(* Logix 5000 project; controller Universal_Device_Info_AOI_V0_1 vendor 1 type 14 code 176 rev 32.11; software revision 32.00; part 10 of 11 *)
(* tags used below, declared in another part *)
   Port : INT;
   Common_Data : Turck_IOLink_Common_Data;
   Write_Application_Specific_Tag : BOOL;
   Universal_IOLink_Info : Universal_IOLink_Info;
   StartupDone : BOOL;
   Done : DINT;
   Error : DINT;
   Active : DINT;
   Pending : DINT;
   Pending_or_Active : DINT;
   MyTicketNum : DINT[32];
   Read_ONS : DINT;
   ReadRequest : DINT;
   Read : DINT;
   DoneCount : DINT;
   Status : DINT;
   ErrorCount : DINT;
   Update_Data : BOOL;
   Write_ONS : DINT;
   WriteRequest : DINT;
(* Universal_Device_Info, continued *)

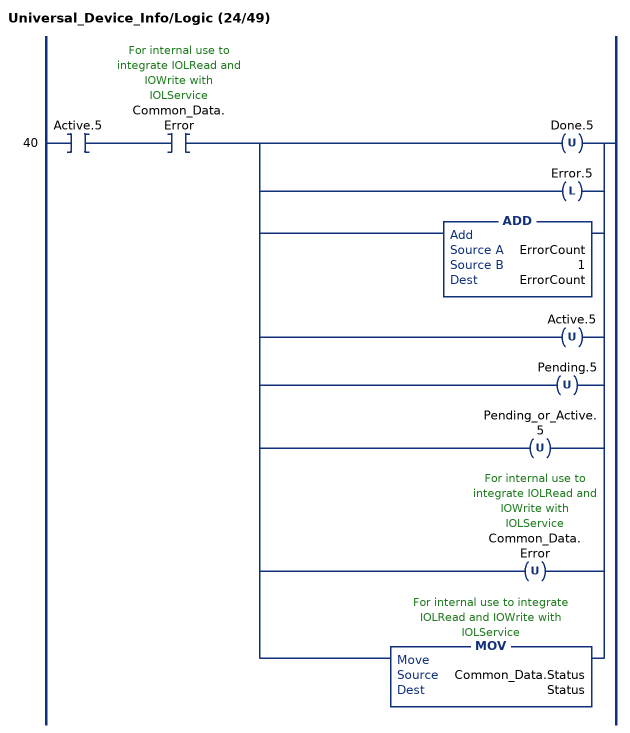
   [picture p67: Universal_Device_Info/Logic rungs 40-40]
   40: XIC(Active.5)XIC(Common_Data.Error)[OTU(Done.5) ,OTL(Error.5) ,ADD(ErrorCount,1,ErrorCount) ,OTU(Active.5) ,OTU(Pending.5) ,OTU(Pending_or_Active.5) ,OTU(Common_Data.Error) ,MOV(Common_Data.Status,Status) ];
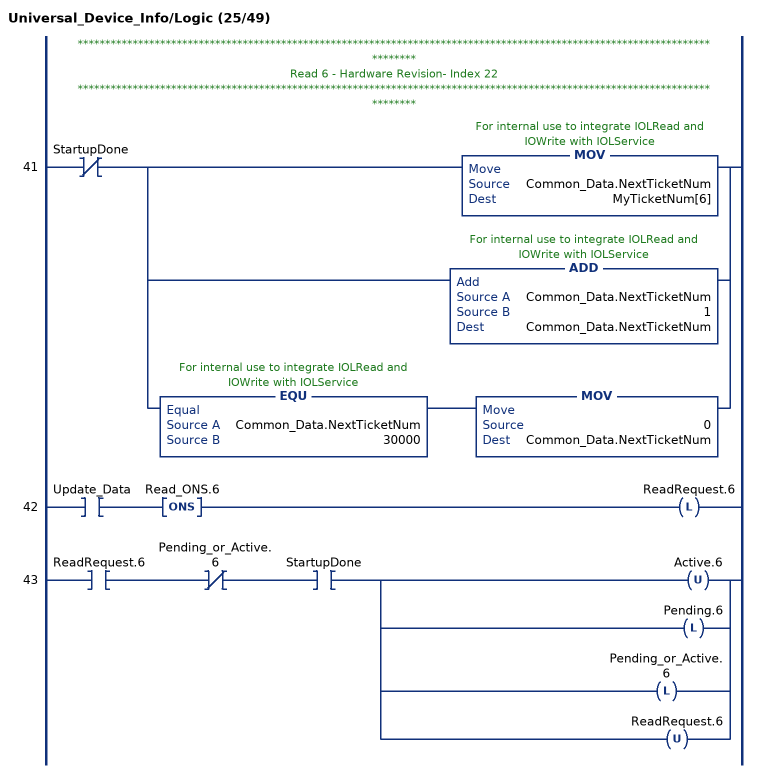
   // ***************************************************************************************************************************
   // Read 6 - Hardware Revision- Index 22
   // ***************************************************************************************************************************
   41: XIO(StartupDone)[MOV(Common_Data.NextTicketNum,MyTicketNum[6]) ,ADD(Common_Data.NextTicketNum,1,Common_Data.NextTicketNum) ,EQU(Common_Data.NextTicketNum,30000) MOV(0,Common_Data.NextTicketNum) ];
   42: XIC(Update_Data)ONS(Read_ONS.6)OTL(ReadRequest.6);
   43: XIC(ReadRequest.6)XIO(Pending_or_Active.6)XIC(StartupDone)[OTU(Active.6) ,OTL(Pending.6) ,OTL(Pending_or_Active.6) ,OTU(ReadRequest.6) ];
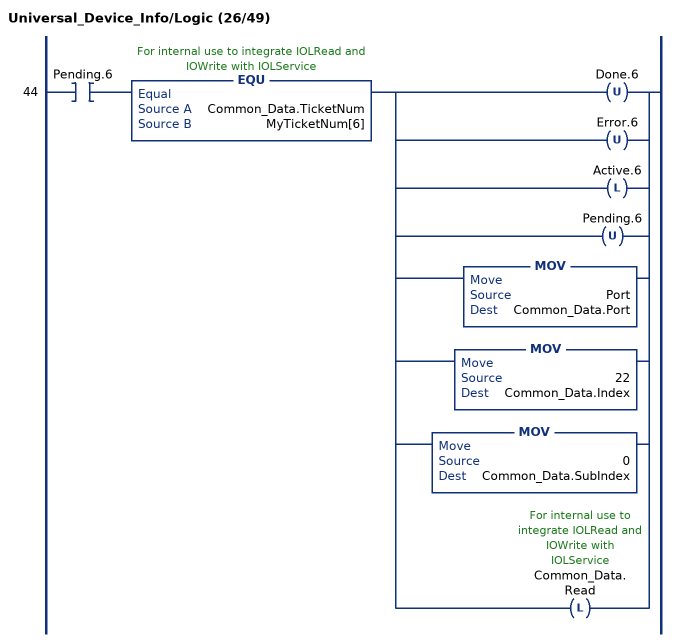
   44: XIC(Pending.6)EQU(Common_Data.TicketNum,MyTicketNum[6])[OTU(Done.6) ,OTU(Error.6) ,OTL(Active.6) ,OTU(Pending.6) ,MOV(Port,Common_Data.Port) ,MOV(22,Common_Data.Index) ,MOV(0,Common_Data.SubIndex) ,OTL(Common_Data.Read) ];
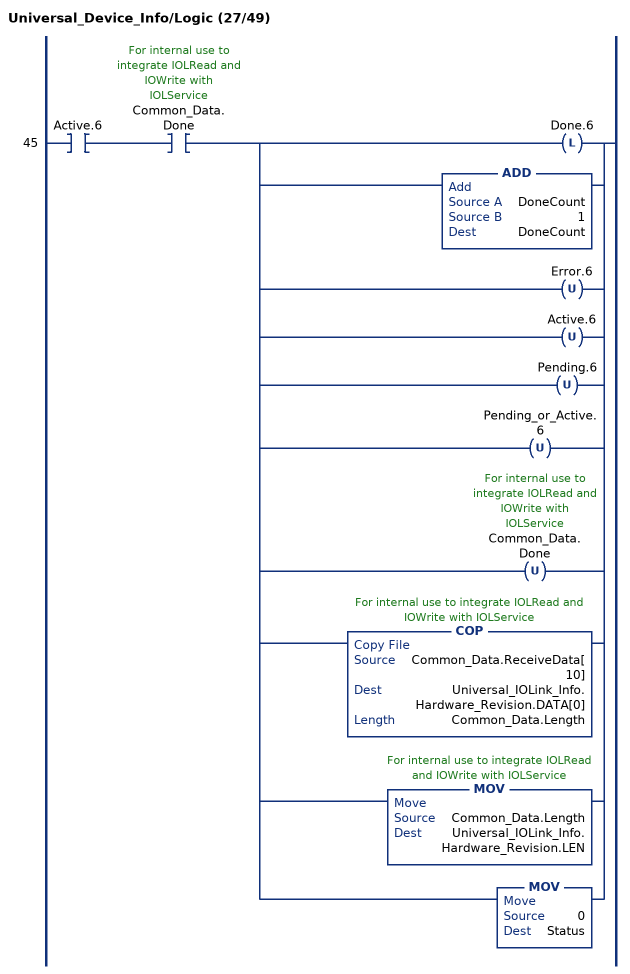
   45: XIC(Active.6)XIC(Common_Data.Done)[OTL(Done.6) ,ADD(DoneCount,1,DoneCount) ,OTU(Error.6) ,OTU(Active.6) ,OTU(Pending.6) ,OTU(Pending_or_Active.6) ,OTU(Common_Data.Done) ,COP(Common_Data.ReceiveData[10],Universal_IOLink_Info.Hardware_Revision.DATA[0],Common_Data.Length) ,MOV(Common_Data.Length,Universal_IOLink_Info.Hardware_Revision.LEN) ,MOV(0,Status) ];
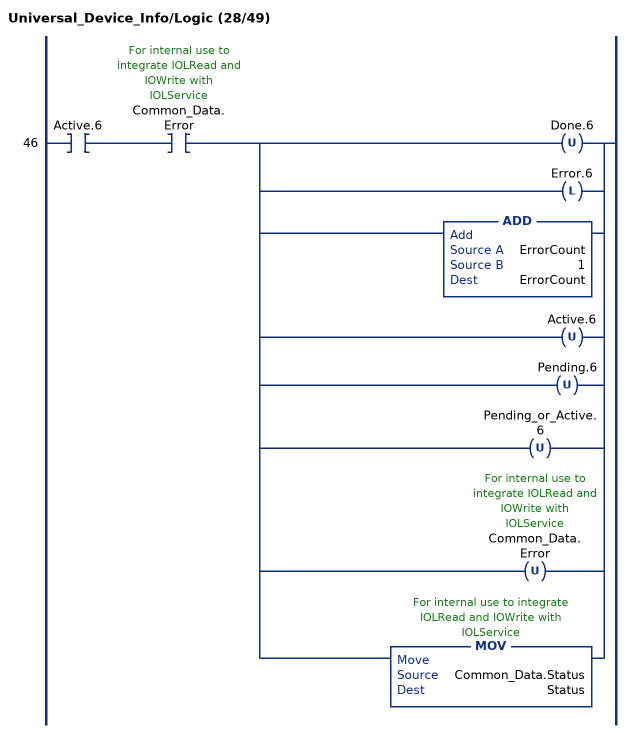
   46: XIC(Active.6)XIC(Common_Data.Error)[OTU(Done.6) ,OTL(Error.6) ,ADD(ErrorCount,1,ErrorCount) ,OTU(Active.6) ,OTU(Pending.6) ,OTU(Pending_or_Active.6) ,OTU(Common_Data.Error) ,MOV(Common_Data.Status,Status) ];
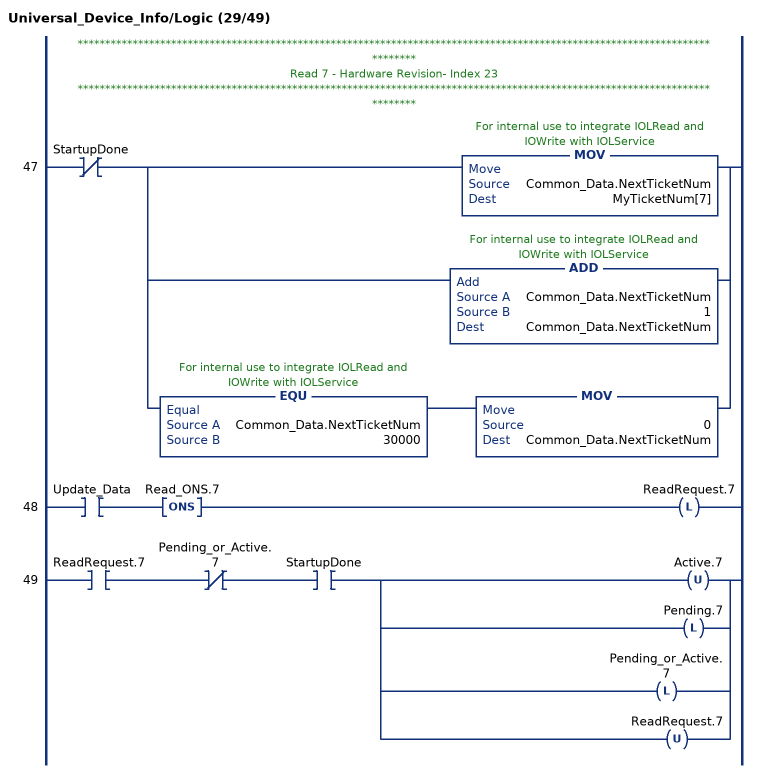
   // ***************************************************************************************************************************
   // Read 7 - Hardware Revision- Index 23
   // ***************************************************************************************************************************
   47: XIO(StartupDone)[MOV(Common_Data.NextTicketNum,MyTicketNum[7]) ,ADD(Common_Data.NextTicketNum,1,Common_Data.NextTicketNum) ,EQU(Common_Data.NextTicketNum,30000) MOV(0,Common_Data.NextTicketNum) ];
   48: XIC(Update_Data)ONS(Read_ONS.7)OTL(ReadRequest.7);
   49: XIC(ReadRequest.7)XIO(Pending_or_Active.7)XIC(StartupDone)[OTU(Active.7) ,OTL(Pending.7) ,OTL(Pending_or_Active.7) ,OTU(ReadRequest.7) ];
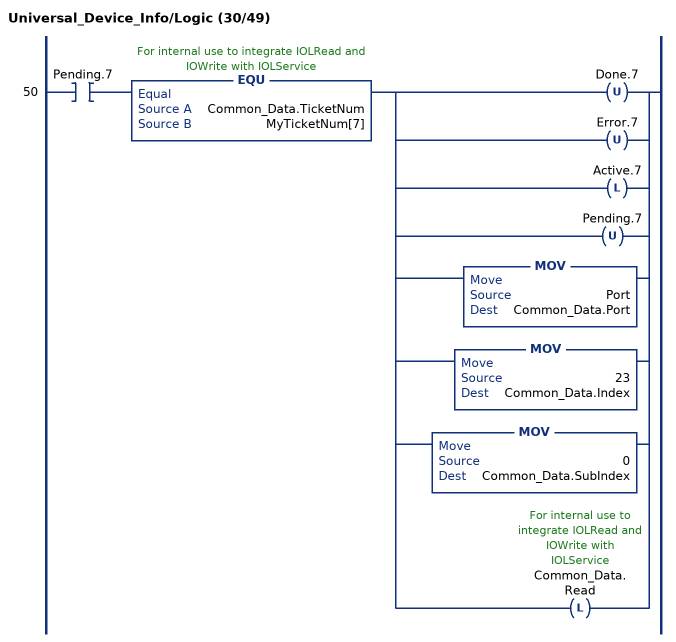
   50: XIC(Pending.7)EQU(Common_Data.TicketNum,MyTicketNum[7])[OTU(Done.7) ,OTU(Error.7) ,OTL(Active.7) ,OTU(Pending.7) ,MOV(Port,Common_Data.Port) ,MOV(23,Common_Data.Index) ,MOV(0,Common_Data.SubIndex) ,OTL(Common_Data.Read) ];
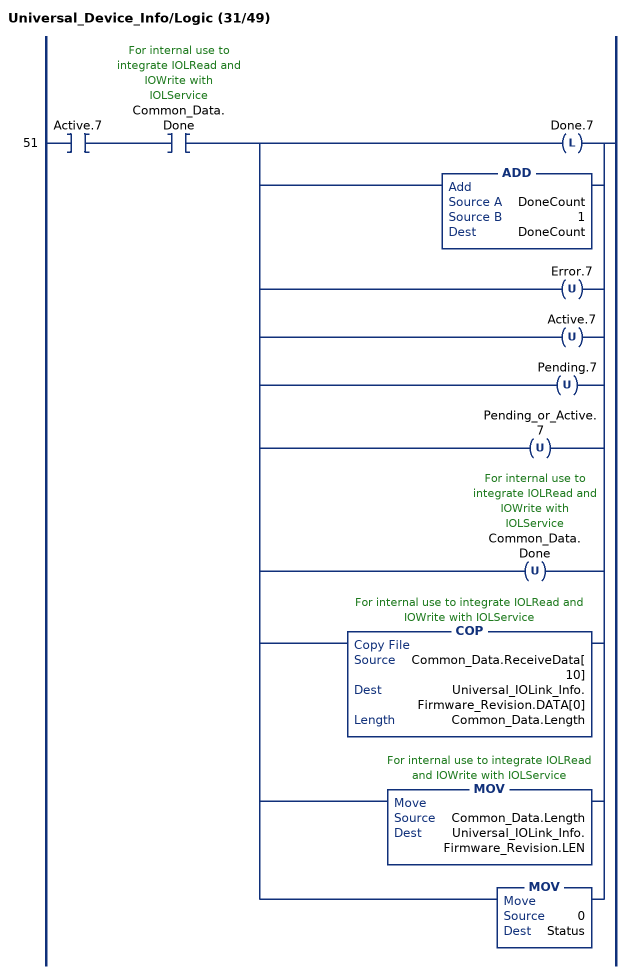
   51: XIC(Active.7)XIC(Common_Data.Done)[OTL(Done.7) ,ADD(DoneCount,1,DoneCount) ,OTU(Error.7) ,OTU(Active.7) ,OTU(Pending.7) ,OTU(Pending_or_Active.7) ,OTU(Common_Data.Done) ,COP(Common_Data.ReceiveData[10],Universal_IOLink_Info.Firmware_Revision.DATA[0],Common_Data.Length) ,MOV(Common_Data.Length,Universal_IOLink_Info.Firmware_Revision.LEN) ,MOV(0,Status) ];
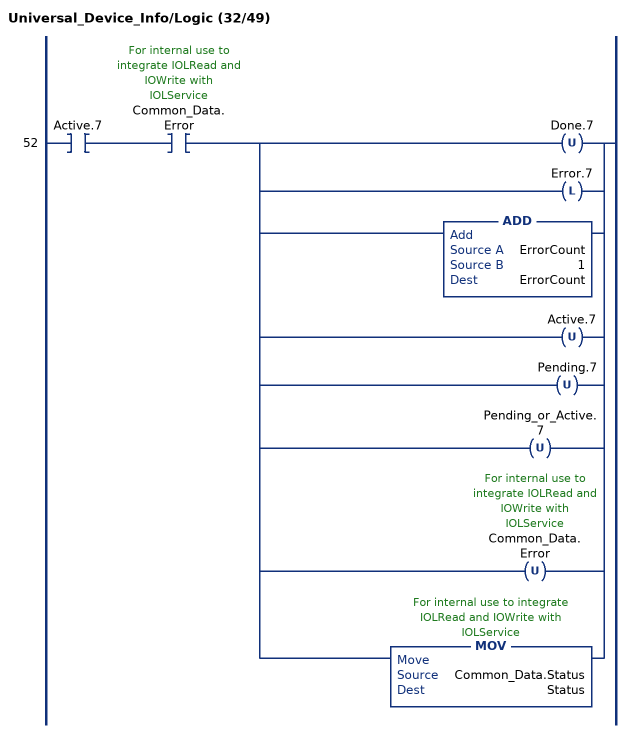
   52: XIC(Active.7)XIC(Common_Data.Error)[OTU(Done.7) ,OTL(Error.7) ,ADD(ErrorCount,1,ErrorCount) ,OTU(Active.7) ,OTU(Pending.7) ,OTU(Pending_or_Active.7) ,OTU(Common_Data.Error) ,MOV(Common_Data.Status,Status) ];
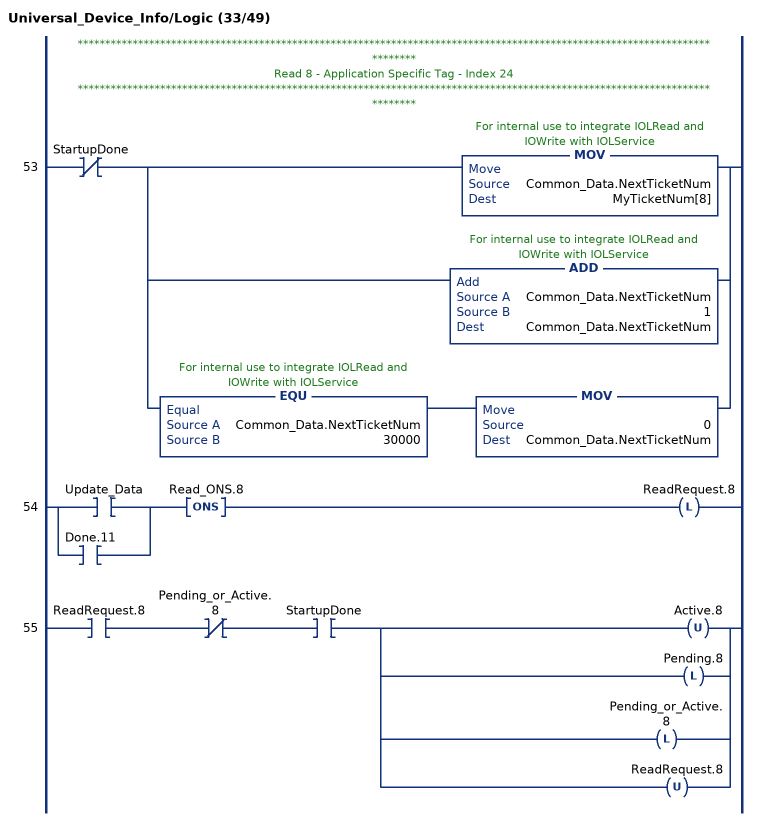
   // ***************************************************************************************************************************
   // Read 8 - Application Specific Tag - Index 24
   // ***************************************************************************************************************************
   53: XIO(StartupDone)[MOV(Common_Data.NextTicketNum,MyTicketNum[8]) ,ADD(Common_Data.NextTicketNum,1,Common_Data.NextTicketNum) ,EQU(Common_Data.NextTicketNum,30000) MOV(0,Common_Data.NextTicketNum) ];
   54: [XIC(Update_Data) ,XIC(Done.11) ]ONS(Read_ONS.8)OTL(ReadRequest.8);
   55: XIC(ReadRequest.8)XIO(Pending_or_Active.8)XIC(StartupDone)[OTU(Active.8) ,OTL(Pending.8) ,OTL(Pending_or_Active.8) ,OTU(ReadRequest.8) ];
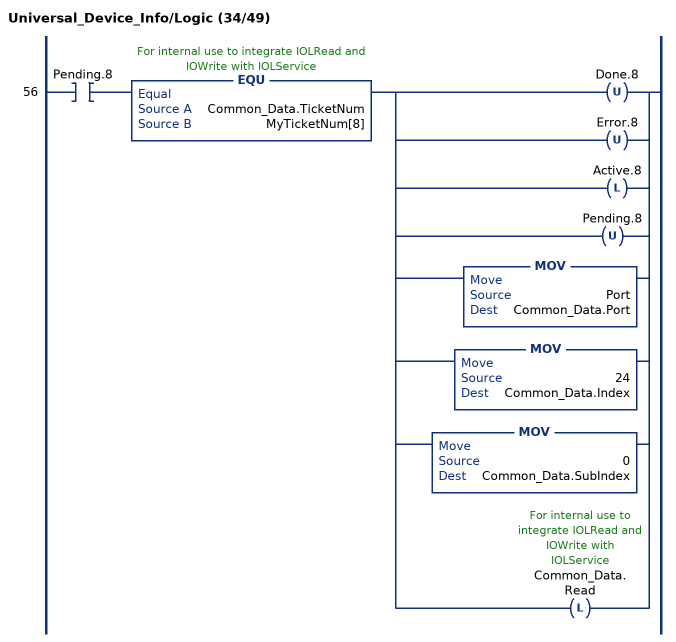
   56: XIC(Pending.8)EQU(Common_Data.TicketNum,MyTicketNum[8])[OTU(Done.8) ,OTU(Error.8) ,OTL(Active.8) ,OTU(Pending.8) ,MOV(Port,Common_Data.Port) ,MOV(24,Common_Data.Index) ,MOV(0,Common_Data.SubIndex) ,OTL(Common_Data.Read) ];
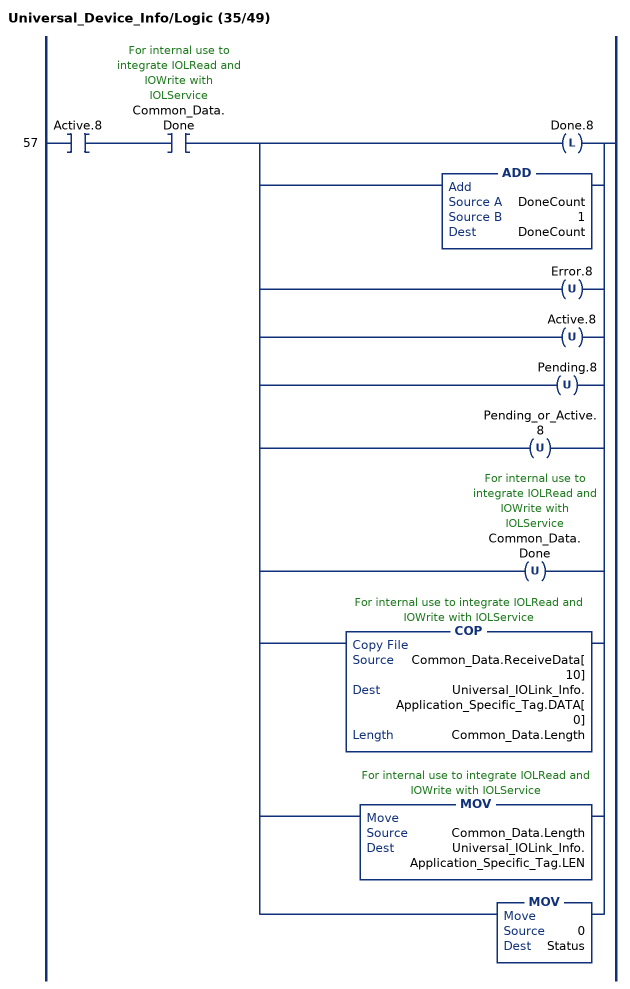
   57: XIC(Active.8)XIC(Common_Data.Done)[OTL(Done.8) ,ADD(DoneCount,1,DoneCount) ,OTU(Error.8) ,OTU(Active.8) ,OTU(Pending.8) ,OTU(Pending_or_Active.8) ,OTU(Common_Data.Done) ,COP(Common_Data.ReceiveData[10],Universal_IOLink_Info.Application_Specific_Tag.DATA[0],Common_Data.Length) ,MOV(Common_Data.Length,Universal_IOLink_Info.Application_Specific_Tag.LEN) ,MOV(0,Status) ];
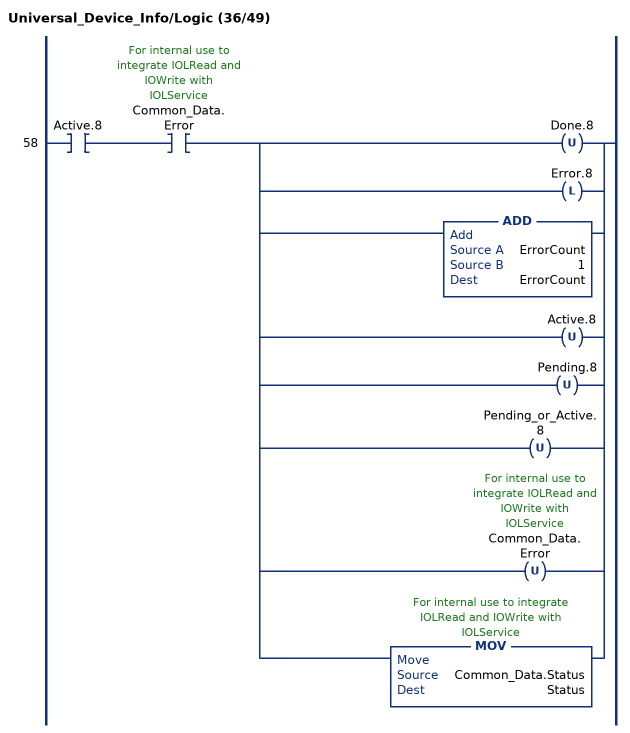
   58: XIC(Active.8)XIC(Common_Data.Error)[OTU(Done.8) ,OTL(Error.8) ,ADD(ErrorCount,1,ErrorCount) ,OTU(Active.8) ,OTU(Pending.8) ,OTU(Pending_or_Active.8) ,OTU(Common_Data.Error) ,MOV(Common_Data.Status,Status) ];
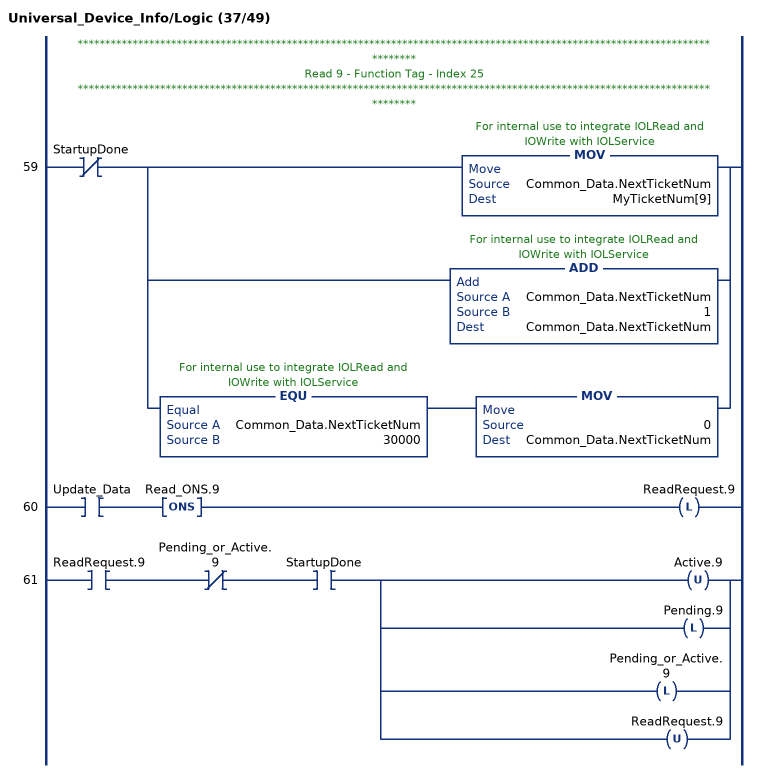
   // ***************************************************************************************************************************
   // Read 9 - Function Tag - Index 25
   // ***************************************************************************************************************************
   59: XIO(StartupDone)[MOV(Common_Data.NextTicketNum,MyTicketNum[9]) ,ADD(Common_Data.NextTicketNum,1,Common_Data.NextTicketNum) ,EQU(Common_Data.NextTicketNum,30000) MOV(0,Common_Data.NextTicketNum) ];
   60: XIC(Update_Data)ONS(Read_ONS.9)OTL(ReadRequest.9);
   61: XIC(ReadRequest.9)XIO(Pending_or_Active.9)XIC(StartupDone)[OTU(Active.9) ,OTL(Pending.9) ,OTL(Pending_or_Active.9) ,OTU(ReadRequest.9) ];
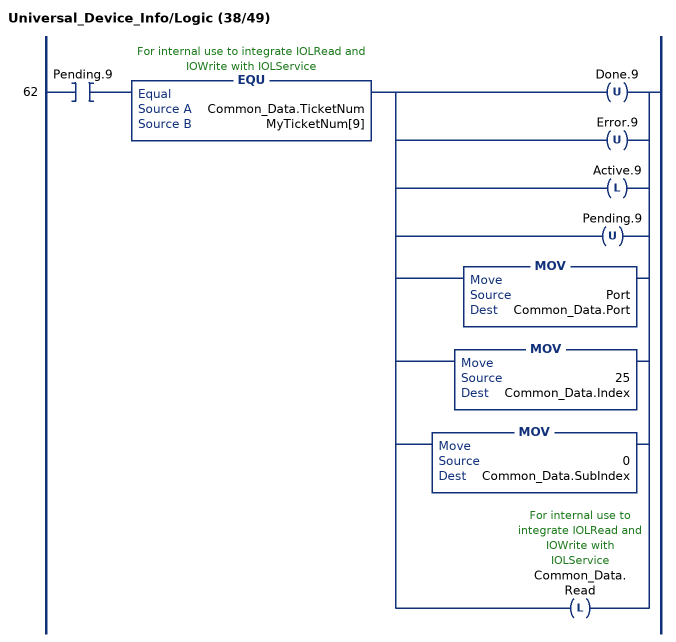
   62: XIC(Pending.9)EQU(Common_Data.TicketNum,MyTicketNum[9])[OTU(Done.9) ,OTU(Error.9) ,OTL(Active.9) ,OTU(Pending.9) ,MOV(Port,Common_Data.Port) ,MOV(25,Common_Data.Index) ,MOV(0,Common_Data.SubIndex) ,OTL(Common_Data.Read) ];
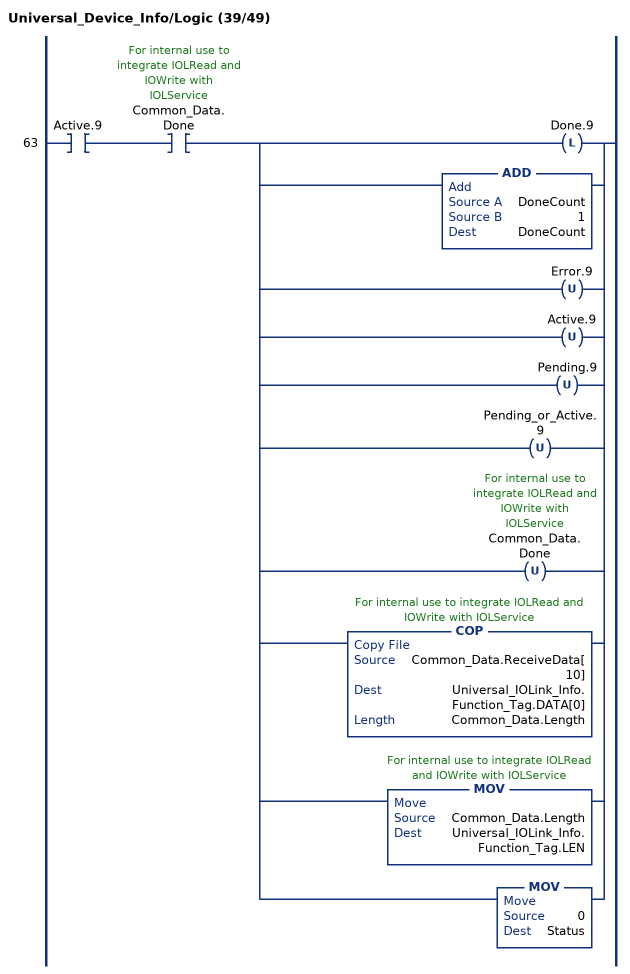
   63: XIC(Active.9)XIC(Common_Data.Done)[OTL(Done.9) ,ADD(DoneCount,1,DoneCount) ,OTU(Error.9) ,OTU(Active.9) ,OTU(Pending.9) ,OTU(Pending_or_Active.9) ,OTU(Common_Data.Done) ,COP(Common_Data.ReceiveData[10],Universal_IOLink_Info.Function_Tag.DATA[0],Common_Data.Length) ,MOV(Common_Data.Length,Universal_IOLink_Info.Function_Tag.LEN) ,MOV(0,Status) ];
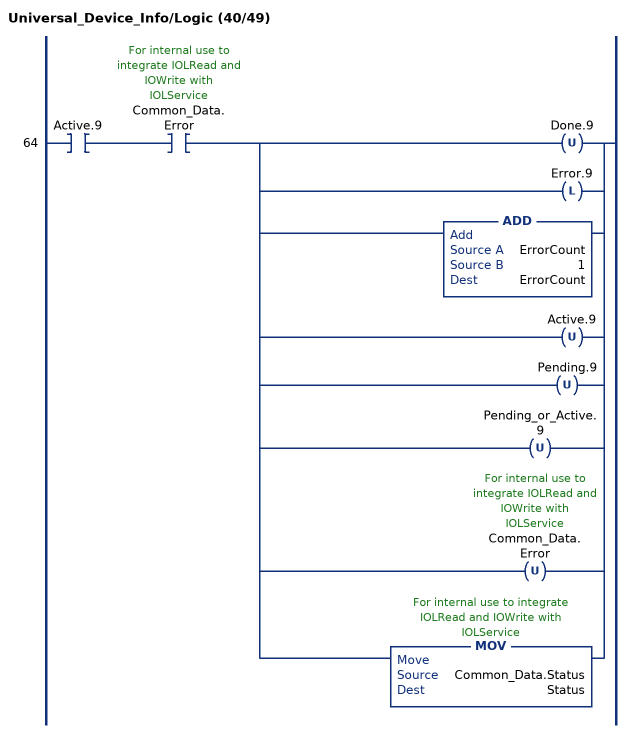
   64: XIC(Active.9)XIC(Common_Data.Error)[OTU(Done.9) ,OTL(Error.9) ,ADD(ErrorCount,1,ErrorCount) ,OTU(Active.9) ,OTU(Pending.9) ,OTU(Pending_or_Active.9) ,OTU(Common_Data.Error) ,MOV(Common_Data.Status,Status) ];
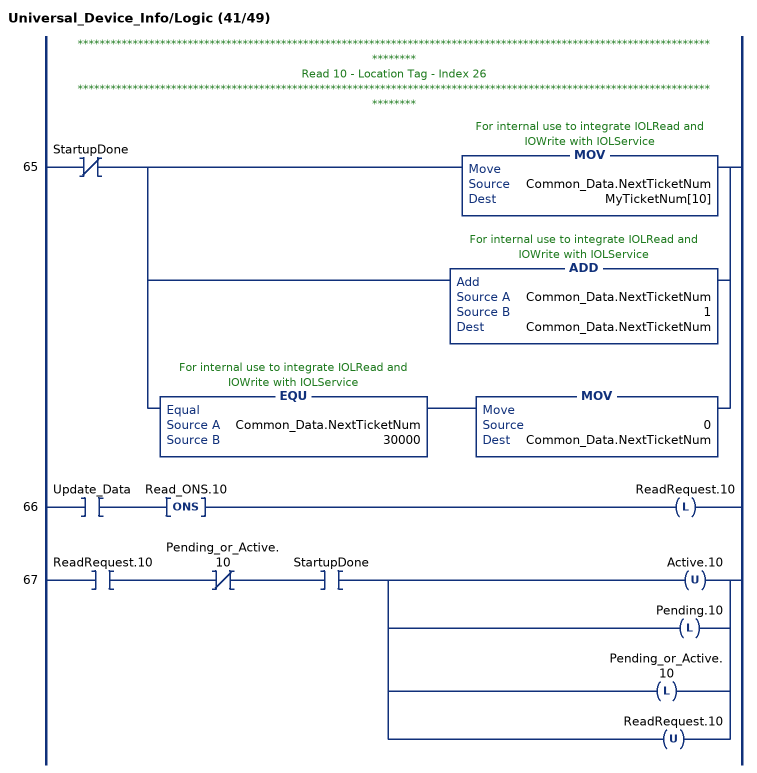
   // ***************************************************************************************************************************
   // Read 10 - Location Tag - Index 26
   // ***************************************************************************************************************************
   65: XIO(StartupDone)[MOV(Common_Data.NextTicketNum,MyTicketNum[10]) ,ADD(Common_Data.NextTicketNum,1,Common_Data.NextTicketNum) ,EQU(Common_Data.NextTicketNum,30000) MOV(0,Common_Data.NextTicketNum) ];
   66: XIC(Update_Data)ONS(Read_ONS.10)OTL(ReadRequest.10);
   67: XIC(ReadRequest.10)XIO(Pending_or_Active.10)XIC(StartupDone)[OTU(Active.10) ,OTL(Pending.10) ,OTL(Pending_or_Active.10) ,OTU(ReadRequest.10) ];
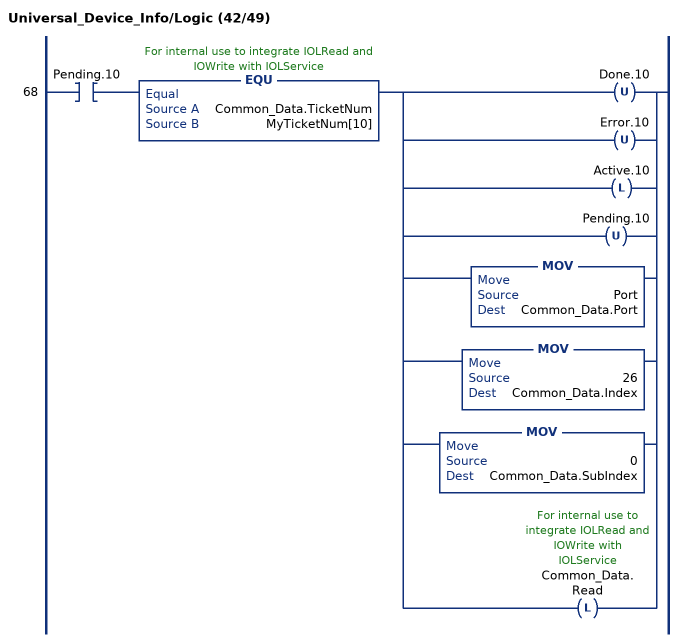
   68: XIC(Pending.10)EQU(Common_Data.TicketNum,MyTicketNum[10])[OTU(Done.10) ,OTU(Error.10) ,OTL(Active.10) ,OTU(Pending.10) ,MOV(Port,Common_Data.Port) ,MOV(26,Common_Data.Index) ,MOV(0,Common_Data.SubIndex) ,OTL(Common_Data.Read) ];
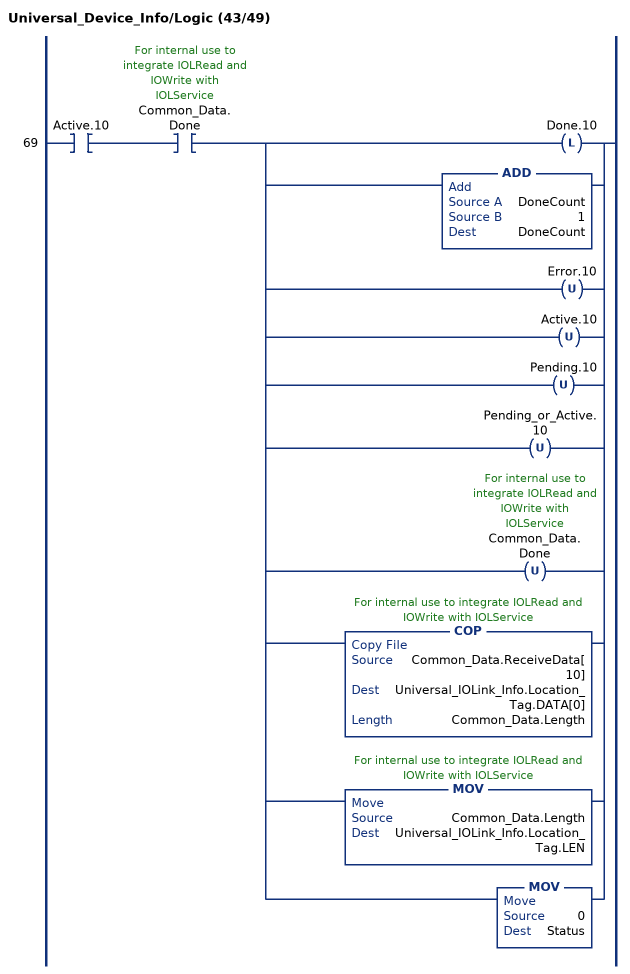
   69: XIC(Active.10)XIC(Common_Data.Done)[OTL(Done.10) ,ADD(DoneCount,1,DoneCount) ,OTU(Error.10) ,OTU(Active.10) ,OTU(Pending.10) ,OTU(Pending_or_Active.10) ,OTU(Common_Data.Done) ,COP(Common_Data.ReceiveData[10],Universal_IOLink_Info.Location_Tag.DATA[0],Common_Data.Length) ,MOV(Common_Data.Length,Universal_IOLink_Info.Location_Tag.LEN) ,MOV(0,Status) ];
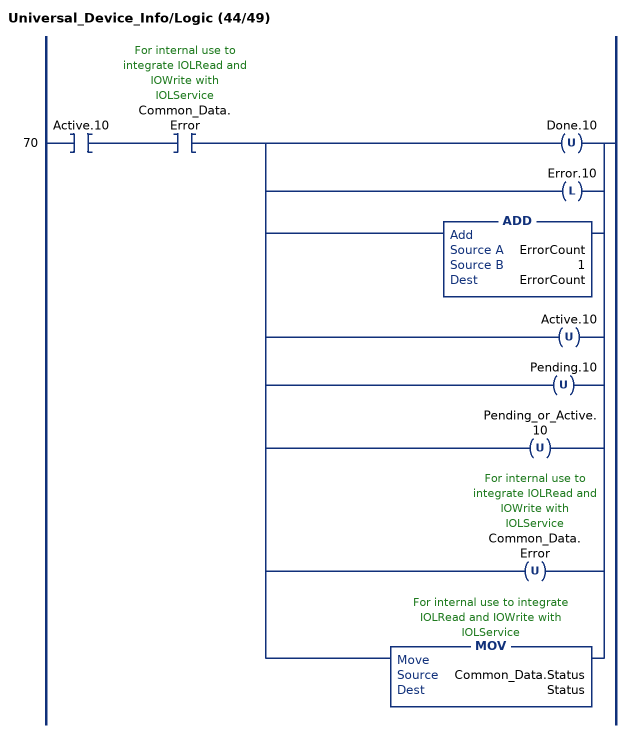
   70: XIC(Active.10)XIC(Common_Data.Error)[OTU(Done.10) ,OTL(Error.10) ,ADD(ErrorCount,1,ErrorCount) ,OTU(Active.10) ,OTU(Pending.10) ,OTU(Pending_or_Active.10) ,OTU(Common_Data.Error) ,MOV(Common_Data.Status,Status) ];
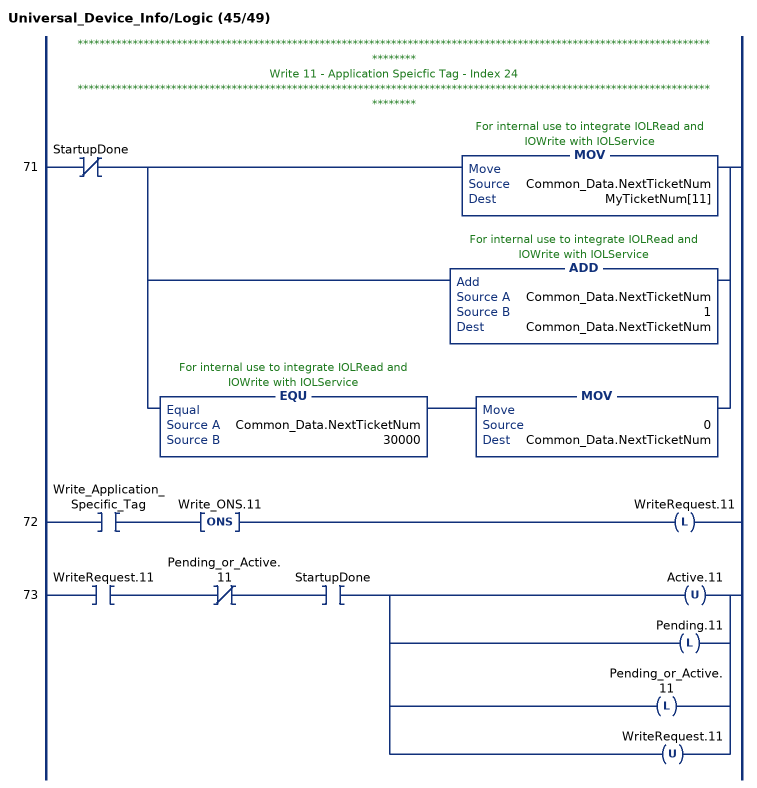
   // ***************************************************************************************************************************
   // Write 11 - Application Speicfic Tag - Index 24
   // ***************************************************************************************************************************
   71: XIO(StartupDone)[MOV(Common_Data.NextTicketNum,MyTicketNum[11]) ,ADD(Common_Data.NextTicketNum,1,Common_Data.NextTicketNum) ,EQU(Common_Data.NextTicketNum,30000) MOV(0,Common_Data.NextTicketNum) ];
   72: XIC(Write_Application_Specific_Tag)ONS(Write_ONS.11)OTL(WriteRequest.11);
   73: XIC(WriteRequest.11)XIO(Pending_or_Active.11)XIC(StartupDone)[OTU(Active.11) ,OTL(Pending.11) ,OTL(Pending_or_Active.11) ,OTU(WriteRequest.11) ];
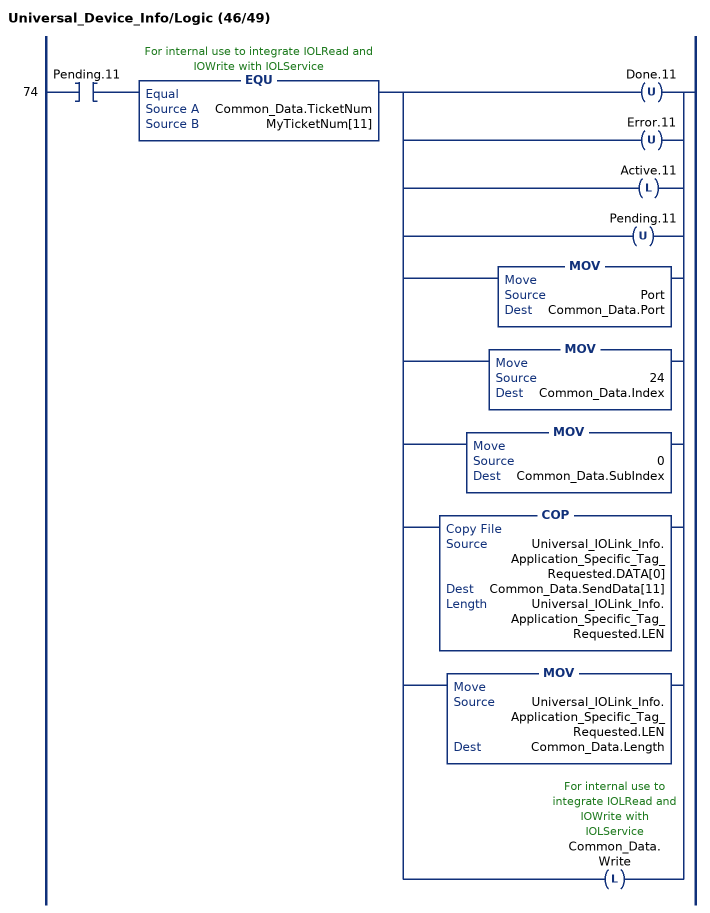
   74: XIC(Pending.11)EQU(Common_Data.TicketNum,MyTicketNum[11])[OTU(Done.11) ,OTU(Error.11) ,OTL(Active.11) ,OTU(Pending.11) ,MOV(Port,Common_Data.Port) ,MOV(24,Common_Data.Index) ,MOV(0,Common_Data.SubIndex) ,COP(Universal_IOLink_Info.Application_Specific_Tag_Requested.DATA[0],Common_Data.SendData[11],Universal_IOLink_Info.Application_Specific_Tag_Requested.LEN) ,MOV(Universal_IOLink_Info.Application_Specific_Tag_Requested.LEN,Common_Data.Length) ,OTL(Common_Data.Write) ];
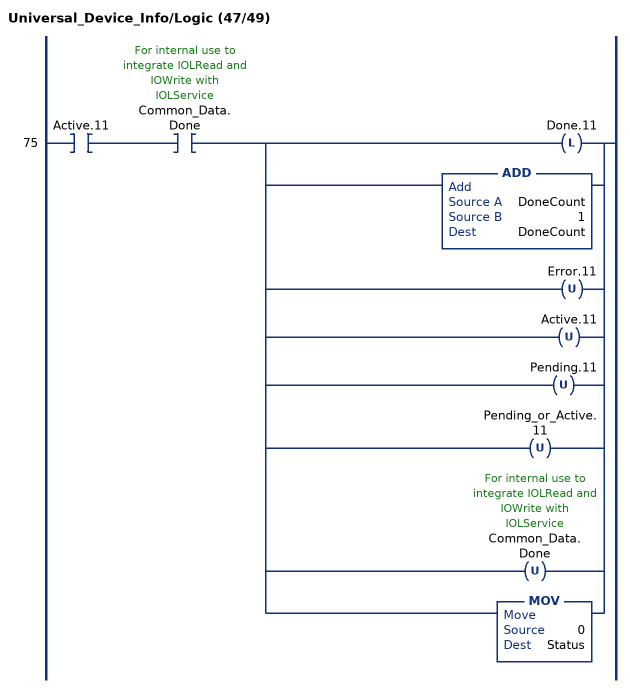
   75: XIC(Active.11)XIC(Common_Data.Done)[OTL(Done.11) ,ADD(DoneCount,1,DoneCount) ,OTU(Error.11) ,OTU(Active.11) ,OTU(Pending.11) ,OTU(Pending_or_Active.11) ,OTU(Common_Data.Done) ,MOV(0,Status) ];
